DATA_BLOCK "AI_Tank5_DB"
{ S7_Optimized_Access := 'FALSE' }
AUTHOR : SimenCom
VERSION : 1.0
"Analog_In_UDT"

BEGIN

END_DATA_BLOCK

